ABB RobotStudio station: FinalProjectStation.rsstn

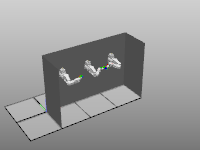
Station FinalProjectStation (saved by RobotStudio 20.4.9280.0)
Controller IRB120Controller_FINALPROJECT
  mechanical unit ROB_1: IRB120_3_58__01, 6 joints, base frame (2400, 0, 1200) mm, rotated rx 0 ry 90 rz -90 deg
  mechanical unit ROB_2: IRB120_3_58__02, 6 joints, base frame (1500, 0, 1200) mm, rotated rx 0 ry 90 rz -90 deg
  mechanical unit ROB_3: IRB120_3_58__03, 6 joints, base frame (600, 0, 1200) mm, rotated rx 0 ry 90 rz -90 deg
Layout (positions relative to the parent item):
  - Wall [part]
  - Smart_Gripper_Servo_Fingers_02 [mechanism, from Tools\ABB_Smart_Gripper_Servo_Fingers.rslib] at (1789.34, -400.57, 1180.86) mm, rotated rx 93.19 ry 0.65 rz 96.19 deg; joint values [0] (rad or m)
  - Smart_Gripper_Servo_Fingers_03 [mechanism, from Tools\ABB_Smart_Gripper_Servo_Fingers.rslib] at (909.26, -560.91, 1195.3) mm, rotated rx 90.72 ry -0.49 rz 124.25 deg; joint values [0] (rad or m)
  - Smart_Gripper_Servo_Fingers_01 [mechanism, from Tools\ABB_Smart_Gripper_Servo_Fingers.rslib] at (2111.95, -340.47, 1186.01) mm, rotated rx -103.75 ry -1.7 rz 110.22 deg; joint values [0] (rad or m)
  - IRB120_3_58__01 [mechanism, from Robots\IRB120_3_58_G_01.rslib] at (2400, 0, 1200) mm, rotated rx 0 ry 90 rz -90 deg; joint values [-1.5848, 0.1047, 1.0175, -0.2544, -1.4723, 0] (rad or m)
  - IRB120_3_58__02 [mechanism, from Robots\IRB120_3_58_G_01.rslib] at (1500, 0, 1200) mm, rotated rx 0 ry 90 rz -90 deg; joint values [1.5014, -0.2054, 0.9237, -0.023, -0.6111, 0] (rad or m)
  - IRB120_3_58__03 [mechanism, from Robots\IRB120_3_58_G_01.rslib] at (600, 0, 1200) mm, rotated rx 0 ry 90 rz -90 deg; joint values [1.5556, -0.2111, 0.2853, 0, 0.5236, 0] (rad or m)
Attachment: Smart_Gripper_Servo_Fingers_01 is attached to IRB120_3_58__01 / Link6
Attachment: Smart_Gripper_Servo_Fingers_02 is attached to IRB120_3_58__02 / Link6
Attachment: Smart_Gripper_Servo_Fingers_03 is attached to IRB120_3_58__03 / Link6
Targets, tools, work objects and paths stored in the station, written as RAPID:
! task T_ROB1
MODULE CalibData
  PERS tooldata Servo:=[TRUE,[[0,0,114.2],[1,0,0,0]],[0.215,[8.7,12.3,49.2],[1,0,0,0],0.00021,0.00024,0.00009]];
ENDMODULE

! task T_ROB2
MODULE CalibData
  PERS tooldata Servo:=[TRUE,[[0,0,114.2],[1,0,0,0]],[0.215,[8.7,12.3,49.2],[1,0,0,0],0.00021,0.00024,0.00009]];
ENDMODULE

! task T_ROB3
MODULE CalibData
  PERS tooldata Servo:=[TRUE,[[0,0,114.2],[1,0,0,0]],[0.215,[8.7,12.3,49.2],[1,0,0,0],0.00021,0.00024,0.00009]];
ENDMODULE

